// SIMATIC S7-200 SMART project (STEP 7-Micro/WIN SMART), CPU CR40

SYMBOL_TABLE 系统符号
Always_On        SM0.0    // 始终接通
First_Scan_On    SM0.1
END_SYMBOL_TABLE

ORGANIZATION_BLOCK MAIN:OB1
TITLE=程序注释
BEGIN
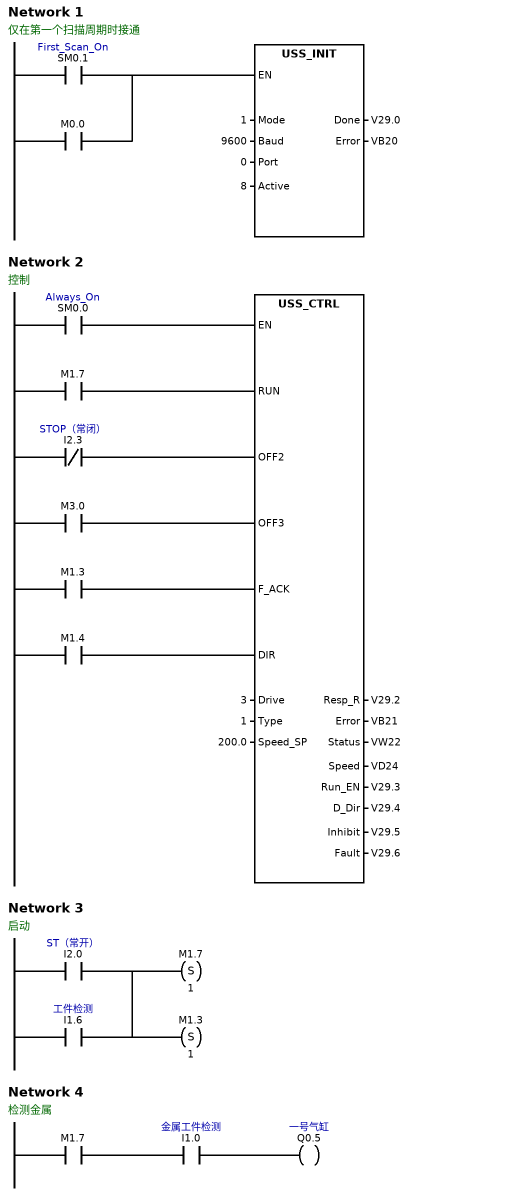
Network 1
// 仅在第一个扫描周期时接通
LD     First_Scan_On:SM0.1
O      M0.0
CALL   USS_INIT:SBR2, 1, 9600, 0, 8, V29.0, VB20
Network 2
// 控制
LD     Always_On:SM0.0
=      L60.0
LD     M1.7
=      L63.7
LDN    STOP（常闭）:I2.3
=      L63.6
LD     M3.0
=      L63.5
LD     M1.3
=      L63.4
LD     M1.4
=      L63.3
LD     L60.0
CALL   USS_CTRL:SBR6, L63.7, L63.6, L63.5, L63.4, L63.3, 3, 1, 200.0, V29.2, VB21, VW22, VD24, V29.3, V29.4, V29.5, V29.6
Network 3
// 启动
LD     ST（常开）:I2.0
O      工件检测:I1.6
S      M1.7, 1
S      M1.3, 1
Network 4
// 检测金属
LD     M1.7
A      金属工件检测:I1.0
=      一号气缸:Q0.5
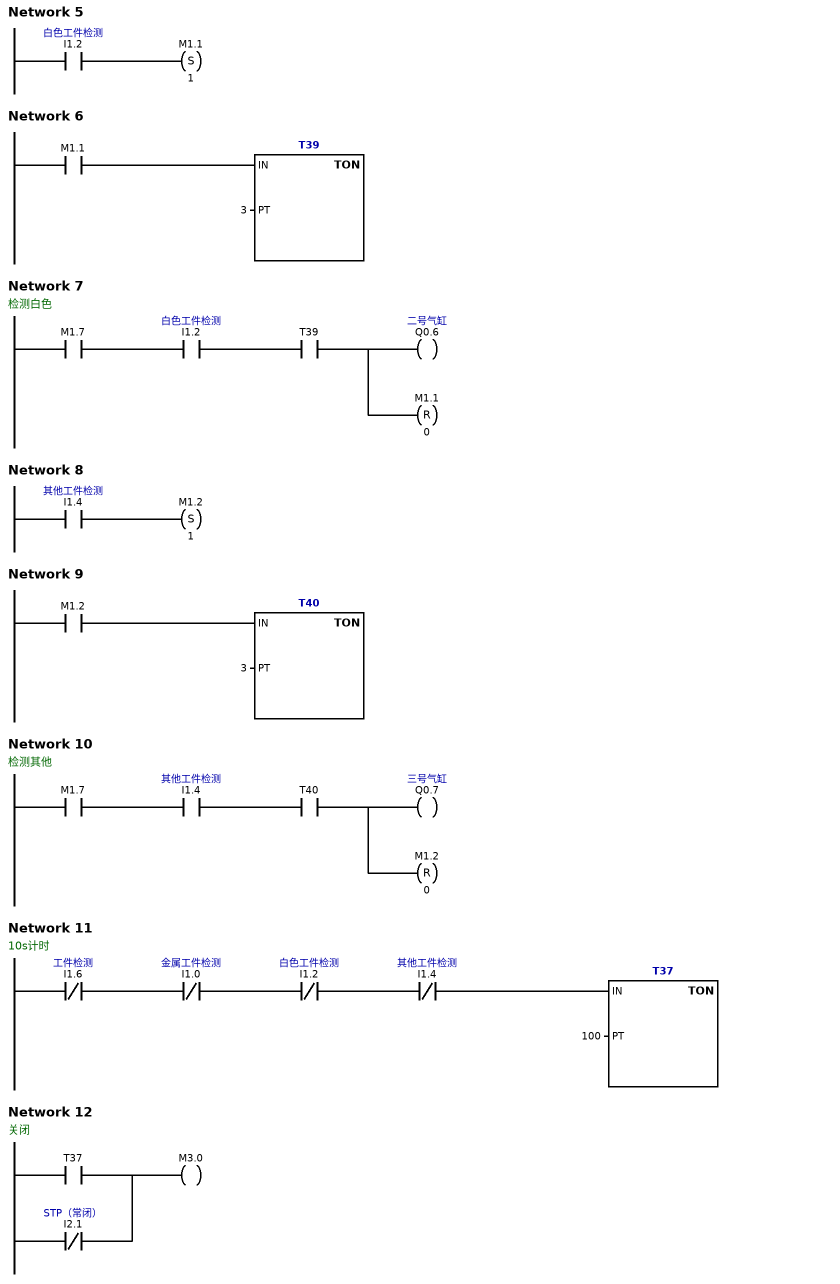
Network 5
LD     白色工件检测:I1.2
S      M1.1, 1
Network 6
LD     M1.1
TON    T39, 3
Network 7
// 检测白色
LD     M1.7
A      白色工件检测:I1.2
A      T39
=      二号气缸:Q0.6
R      M1.1, 0
Network 8
LD     其他工件检测:I1.4
S      M1.2, 1
Network 9
LD     M1.2
TON    T40, 3
Network 10
// 检测其他
LD     M1.7
A      其他工件检测:I1.4
A      T40
=      三号气缸:Q0.7
R      M1.2, 0
Network 11
// 10s计时
LDN    工件检测:I1.6
AN     金属工件检测:I1.0
AN     白色工件检测:I1.2
AN     其他工件检测:I1.4
TON    T37, 100
Network 12
// 关闭
LD     T37
ON     STP（常闭）:I2.1
=      M3.0
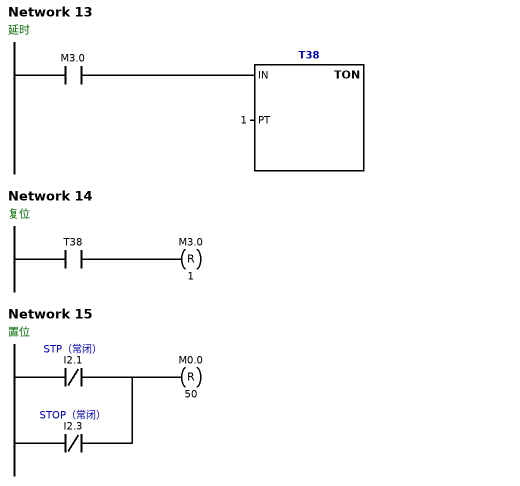
Network 13
// 延时
LD     M3.0
TON    T38, 1
Network 14
// 复位
LD     T38
R      M3.0, 1
Network 15
// 置位
LDN    STP（常闭）:I2.1
ON     STOP（常闭）:I2.3
R      M0.0, 50
END_ORGANIZATION_BLOCK

// SBR2: protected block, not included

// SBR3: protected block, not included

// SBR4: protected block, not included

// SBR5: protected block, not included

// SBR6: protected block, not included

// INT1: protected block, not included
